# EPICS substitutions: ek9000App/Db/EL1088.substitutions
file EL1088.template
{       pattern
        {
                TERMINAL,

        }
        {
        }
}
